INTERFACE I_StringBuilder

// Adds a string to the build sequence.
METHOD AddString : I_StringBuilder
VAR_INPUT
	str	: Tc2_System.T_MaxString;	// String to be added.
END_VAR
END_METHOD

// Finishes string generation and returns the generated string
METHOD Create : Tc2_System.T_MaxString
END_METHOD

// Reset the string build sequence, clear any string built so far. Returns the string builder instance
METHOD Reset	: I_StringBuilder
END_METHOD

END_INTERFACE

(* stored: Version 1.1.0.1, ProductVersion 3.1.4024.13
   Itf I_StringBuilder: Id {3747aab2-3bd3-07b0-2f01-57cd97da3929}
   Method AddString: Id {0ad7aba7-4db1-04cc-1556-52b420102f2c}
   Method Create: Id {c5baa772-95a0-07ec-3a50-e773e513123b}
   Method Reset: Id {5a2a6527-e07d-07ab-15c7-6e9f6a27c164} *)
